// TIA Portal V20 export
FUNCTION_BLOCK "FB_ButtonsLamps"   // FB2, LAD
{ S7_Optimized_Access := 'TRUE' }
// stored: MemoryReserve 100, SetENOAutomatically false
BEGIN

REGION Network 1 (SCL)
   IF "AlwaysTRUE" THEN
       "AlwaysTRUE" := "AlwaysTRUE";
   END_IF;
END_REGION
END_FUNCTION_BLOCK
